TYPE ST_TransferHandshakeSignal :
STRUCT
	Accept : BOOL;
	Ready : BOOL;
	ReceiveRequest : BOOL;
	SendRequest : BOOL;
	SendComplete : BOOL;
	ReceiveComplete : BOOL;
END_STRUCT
END_TYPE

(* stored: Version 1.1.0.1, ProductVersion 3.1.4026.18
   DUT ST_TransferHandshakeSignal: Id {b01d4a3d-ec03-4bfb-ba0a-fd772e348611} *)
